PROGRAM run
VAR
END_VAR

GVL.runner.run(disable_ads_output:=TRUE);

END_PROGRAM

(* stored: Version 1.1.0.1, ProductVersion 3.1.4024.9
   POU run: Id {05dbd5a8-7a86-47ce-bc01-832a4b36dd53}, SpecialFunc None *)
